Universal Robots PolyScope program: test_gripper.urp

Program test_gripper (installation=default directory=/programs/new folder_2 createdIn=5.11.9.1010452 lastSavedIn=5.11.9.1010452 robotSerialNumber=20225200364)
Calibrated DH parameters: a=[0.00002, -0.569483, -0.54992, -0.00001, -0.000036, 0]; d=[0.180894, -146.691669, 192.918669, -46.053088, 0.119778, 0.115602]; alpha=[1.571425, -0.001534, 0.003359, 1.568739, -1.571477, 0]; deltaTheta=[0, 0.376258, -0.101074, -0.275185, -0.000002, 0]
Robot Program (runOnlyOnce=false)
  Script file /programs/usbdisk/Industrial_Centre/ICLTC_MASSAGE_ROBOT/Test_Gripper.script
    | # ============================================================
    | # MINIMAL: UR10e + OnRobot RG2V2 via XML-RPC (localhost:41414)
    | # No RTDE architecture. Import as .script and run.
    | # Motion: 20cm straight line, rhythmic grip: CLOSE -> OPEN -> MOVE
    | # ============================================================
    | 
    | # ---------- User parameters ----------
    | A_SLOW = 0.40
    | V_SLOW = 0.05
    | R_BLEND = 0.005
    | 
    | LINE_LEN_M = 0.20
    | N_STEPS = 10
    | DWELL_S = 0.15
    | 
    | # Direction in BASE frame (default +Y)
    | DIR_X = 0.0
    | DIR_Y = 1.0
    | DIR_Z = 0.0
    | 
    | # RG2V2 parameters (RG2: width 0..110 mm, force up to 40 N)
    | RG_TOOL_INDEX = 0
    | RG_CLOSE_WIDTH_MM = 0.0
    | RG_OPEN_WIDTH_MM  = 110.0
    | RG_FORCE_N = 40.0
    | 
    | # ---------- OnRobot Tool Communication + XML-RPC ----------
    | # These settings match what your generated script uses.
    | set_tool_voltage(24)
    | set_tool_communication(True, 1000000, 2, 1, 1.5, 3.5)
    | 
    | # OnRobot URCap local RPC endpoint (from your generated script)
    | on_tool_xmlrpc = rpc_factory("xmlrpc", "http://localhost:41414")
    | 
    | def rg2_grip(width_mm, force_n):
    |   # width_mm: 0..110 (RG2)
    |   # force_n : 0..40  (RG2)
    |   local ret = on_tool_xmlrpc.rg_grip(RG_TOOL_INDEX, width_mm + 0.0, force_n + 0.0)
    |   if (ret != 0):
    |     popup("OnRobot rg_grip() returned error: " + to_str(ret), title="RG2 Error", error=True, blocking=False)
    |     halt
    |   end
    | end
    | 
    | def gripper_close():
    |   rg2_grip(RG_CLOSE_WIDTH_MM, RG_FORCE_N)
    |   sleep(DWELL_S)
    | end
    | 
    | def gripper_open():
    |   rg2_grip(RG_OPEN_WIDTH_MM, RG_FORCE_N)
    |   sleep(DWELL_S)
    | end
    | 
    | # ---------- Main ----------
    | start_pose = get_actual_tcp_pose()
    | rx = start_pose[3]
    | ry = start_pose[4]
    | rz = start_pose[5]
    | 
    | if (N_STEPS < 1):
    |   N_STEPS = 1
    | end
    | step = LINE_LEN_M / N_STEPS
    | 
    | textmsg("RG2 minimal demo start. steps=", N_STEPS)
    | 
    | # optional: start from open
    | gripper_open()
    | 
    | i = 0
    | while (i <= N_STEPS):
    | 
    |   # rhythm
    |   gripper_close()
    |   gripper_open()
    | 
    |   # straight move
    |   target = p[
    |     start_pose[0] + (i * step) * DIR_X,
    |     start_pose[1] + (i * step) * DIR_Y,
    |     start_pose[2] + (i * step) * DIR_Z,
    |     rx, ry, rz
    |   ]
    | 
    |   movel(target, a=A_SLOW, v=V_SLOW, r=R_BLEND)
    | 
    |   i = i + 1
    | end
    | 
    | gripper_open()
    | textmsg("RG2 minimal demo done.")
  Halt
